TYPE "UDT_Word"
VERSION : 0.1
// Block: UDT_Word
   STRUCT
      b_0 : Bool;
      b_1 : Bool;
      b_2 : Bool;
      b_3 : Bool;
      b_4 : Bool;
      b_5 : Bool;
      b_6 : Bool;
      b_7 : Bool;
      b_8 : Bool;
      b_9 : Bool;
      b_10 : Bool;
      b_11 : Bool;
      b_12 : Bool;
      b_13 : Bool;
      b_14 : Bool;
      b_15 : Bool;
   END_STRUCT;

END_TYPE
